(* IEC 61131-3 sources: repolevel_ST_code_completion/extract_code/重型运输系统/can/FUN, 13 files *)

(* ---- CAN_Read_Data_SWMC.st ---- *)
FUNCTION CAN_Read_Data_SWMC : Can_baseframe
VAR_INPUT
	SWMC_ID	 :UINT;		//接收SWMC控制ID
	I	 	 :UINT;      //接收缓冲区域
END_VAR
VAR
	frame :Can_baseframe;
END_VAR

CASE  SWMC_ID OF

	1:                       //SWMC-C1
		frame.id 	:= (gCan.C1RxMsg.RXMsg[I].RxMsg_CobId-8)/32;
		frame.data 	:= gCan.C1RxMsg.RXMsg[I].RxMsg_Byte;
	2:                       //SWMC-C2
		frame.id 	:= (gCan.C2RxMsg.RXMsg[I].RxMsg_CobId-8)/32;
		frame.data 	:= gCan.C2RxMsg.RXMsg[I].RxMsg_Byte;
	3:						//SWMC-C3
		frame.id 	:= (gCan.C3RxMsg.RXMsg[I].RxMsg_CobId-8)/32;
		frame.data 	:= gCan.C3RxMsg.RXMsg[I].RxMsg_Byte;
	4:                       //SWMC-C4
		frame.id 	:= (gCan.C4RxMsg.RXMsg[I].RxMsg_CobId-8)/32;
		frame.data 	:= gCan.C4RxMsg.RXMsg[I].RxMsg_Byte;
	//(*
	5:                       //SWMC-C5
		frame.id 	:= (gCan.C5RxMsg.RXMsg[I].RxMsg_CobId-8)/32;
		frame.data 	:= gCan.C5RxMsg.RXMsg[I].RxMsg_Byte;
	6:						//SWMC-C6
		frame.id 	:= (gCan.C6RxMsg.RXMsg[I].RxMsg_CobId-8)/32;
		frame.data 	:= gCan.C6RxMsg.RXMsg[I].RxMsg_Byte;
		//*)
	ELSE				//Other
		frame.id := 0;
		frame.data[1] := 0;
		frame.data[2] := 0;
		frame.data[3] := 0;
		frame.data[4] := 0;
		frame.data[5] := 0;
		frame.data[6] := 0;
		frame.data[7] := 0;
		frame.data[8] := 0;
END_CASE
Can_Read_data_SWMC := frame;

(* ---- CAN_Send_Data_SWMC.st ---- *)
FUNCTION CAN_Send_Data_SWMC : BOOL
VAR_INPUT
	SWMC_ID : UINT;
	id 		: UINT;
	data	: ARRAY[1..8] OF BYTE;
END_VAR
VAR

END_VAR

CASE  SWMC_ID OF

	1:
		gCan.C1TxMsg.TXMsg[1].TxMsg_CobId 	:= 8 + 32 * id;
	  	gCan.C1TxMsg.TXMsg[1].TxMsg_Byte 	:= data;
	   	gCan.C1TxMsg.NoOfTxMessages			:= 1;
	   	gCan.C1TxMsg.TxCounter 				:= gCan.C1TxMsg.TxCounter +1;
	2:
		gCan.C2TxMsg.TXMsg[1].TxMsg_CobId 	:= 8 + 32 * id;
	  	gCan.C2TxMsg.TXMsg[1].TxMsg_Byte 	:= data;
	   	gCan.C2TxMsg.NoOfTxMessages			:= 1;
	   	gCan.C2TxMsg.TxCounter 				:= gCan.C2TxMsg.TxCounter +1;
	3:
		gCan.C3TxMsg.TXMsg[1].TxMsg_CobId 	:= 8 + 32 * id;
	  	gCan.C3TxMsg.TXMsg[1].TxMsg_Byte 	:= data;
	   	gCan.C3TxMsg.NoOfTxMessages			:= 1;
	   	gCan.C3TxMsg.TxCounter 				:= gCan.C3TxMsg.TxCounter +1;
	4:
		gCan.C4TxMsg.TXMsg[1].TxMsg_CobId 	:= 8 + 32 * id;
	  	gCan.C4TxMsg.TXMsg[1].TxMsg_Byte 	:= data;
	   	gCan.C4TxMsg.NoOfTxMessages			:= 1;
	   	gCan.C4TxMsg.TxCounter 				:= gCan.C4TxMsg.TxCounter +1;
	//(*
	5:
		gCan.C5TxMsg.TXMsg[1].TxMsg_CobId 	:= 8 + 32 * id;
	  	gCan.C5TxMsg.TXMsg[1].TxMsg_Byte 	:= data;
	   	gCan.C5TxMsg.NoOfTxMessages			:= 1;
	   	gCan.C5TxMsg.TxCounter 				:= gCan.C5TxMsg.TxCounter +1;
	6:
		gCan.C6TxMsg.TXMsg[1].TxMsg_CobId 	:= 8 + 32 * id;
	  	gCan.C6TxMsg.TXMsg[1].TxMsg_Byte 	:= data;
	   	gCan.C6TxMsg.NoOfTxMessages			:= 1;
	   	gCan.C6TxMsg.TxCounter 				:= gCan.C6TxMsg.TxCounter +1;
	//*)

END_CASE

(* ---- percentCalc.st ---- *)
FUNCTION percentCalc : REAL
VAR_INPUT
	level		:INT;	//1->地轨	2->天轨
	idx			:INT;	//挡板索引编号
END_VAR
VAR
	c			:REAL;
	p			:REAL;
END_VAR

//伸出百分比计算
CASE level OF
	1:
		IF gDev.grd[idx].sensor.position < 3 THEN
			RETURN;
		END_IF
		c := gDev.grd[idx].sensor.position - gDev.grd[idx].sensor.retractVal;
		p := gDev.grd[idx].sensor.extendVal - gDev.grd[idx].sensor.retractVal;
		percentCalc := c * 100 / p;
	2:
		IF gDev.sky[idx].sensor.position < 3 THEN
			RETURN;
		END_IF
		c := gDev.sky[idx].sensor.position - gDev.sky[idx].sensor.retractVal;
		p := gDev.sky[idx].sensor.extendVal - gDev.sky[idx].sensor.retractVal;
		percentCalc := c * 100 / p;
END_CASE

(* ---- setButtonByDirect.st ---- *)
FUNCTION setButtonByDirect : BOOL
VAR_INPUT
	level		:INT;	//1->地轨	2->天轨
	idx			:INT;	//挡板索引编号
	direct		:TargetDirect;
END_VAR
VAR
END_VAR
//	本函数用于根据输入参数 操作UI界面的按钮变量
CASE level OF
	1:
		IF idx = 0 OR idx > 10 THEN		//参数校验
			RETURN;
		END_IF
		CASE direct OF
			TargetDirect.extend:
				gUI.grd[idx].btnStop := FALSE;
				gUI.grd[idx].btnExtend := TRUE;
				gUI.grd[idx].btnRetract := FALSE;
			TargetDirect.retract:
				gUI.grd[idx].btnStop := FALSE;
				gUI.grd[idx].btnExtend := FALSE;
				gUI.grd[idx].btnRetract := TRUE;
			TargetDirect.stop:
				gUI.grd[idx].btnStop := FALSE;
				gUI.grd[idx].btnExtend := FALSE;
				gUI.grd[idx].btnRetract := FALSE;
		END_CASE
	2:
		IF idx > 10 THEN		//参数校验
			RETURN;
		END_IF
		CASE direct OF
			TargetDirect.extend:
				gUI.sky[idx].btnStop := FALSE;
				gUI.sky[idx].btnExtend := TRUE;
				gUI.sky[idx].btnRetract := FALSE;
			TargetDirect.retract:
				gUI.sky[idx].btnStop := FALSE;
				gUI.sky[idx].btnExtend := FALSE;
				gUI.sky[idx].btnRetract := TRUE;
			TargetDirect.stop:
				gUI.sky[idx].btnStop := FALSE;
				gUI.sky[idx].btnExtend := FALSE;
				gUI.sky[idx].btnRetract := FALSE;
		END_CASE

END_CASE;

(* ---- updateDevStatus.st ---- *)
FUNCTION updateDevStatus : DevStatus
VAR_INPUT
	level		:INT;		//1->地轨	2->天轨
	idx			:INT;		//挡板索引编号
	errorVal	:REAL;		//误差范围
END_VAR
VAR
	extendVal	:REAL;		//伸出值
	retractVal	:REAL;		//缩回到位值
	nowVal		:REAL;		//当前值
	stat		:DevStatus;	//设备状态
END_VAR

(* 本函数用于根据设备的标定伸出/缩回值以及当前位置
** 判断该缸体是否处于伸出/缩回到位状态，如果到位更新参数
*)

stat := DevStatus.unknown;	//初始化状态量
CASE level OF
	1:
		extendVal := gDev.grd[idx].sensor.extendVal;
		retractVal := gDev.grd[idx].sensor.retractVal;
		nowVal := gDev.grd[idx].sensor.position;
		stat := gDev.grd[idx].state;
	2:
		extendVal := gDev.sky[idx].sensor.extendVal;
		retractVal := gDev.sky[idx].sensor.retractVal;
		nowVal := gDev.sky[idx].sensor.position;
		stat := gDev.sky[idx].state;
END_CASE

IF nowVal > 1 THEN
	IF nowVal < retractVal + errorVal THEN
		stat := DevStatus.retracted;
	ELSIF nowVal > extendVal - errorVal THEN
		stat := DevStatus.extended;
	ELSE
		IF stat <> DevStatus.runing THEN
			stat := DevStatus.error;
		END_IF
	END_IF
ELSE
	stat := DevStatus.unknown;
END_IF

CASE level OF
	1:
		gDev.grd[idx].state := stat;
	2:
		gDev.sky[idx].state := stat;
END_CASE

updateDevStatus := stat;

(* ---- CommandExecutor.st ---- *)
FUNCTION_BLOCK CommandExecutor
VAR_INPUT
	level		:INT;			//1->地轨	2->天轨
	idx			:INT;			//挡板索引编号
	percent		:REAL;			//比例阀百分比 传入-100~+100
END_VAR
VAR_OUTPUT
END_VAR
VAR
END_VAR

IF percent > 0 THEN
	CASE level OF
		1:
			gController.grd[idx].extendPercent := REAL_TO_WORD(percent * 65535 / 100);
			gController.grd[idx].retractPercent := 0;
		2:
			gController.sky[idx].extendPercent := REAL_TO_WORD(percent * 65535 / 100);
			gController.sky[idx].retractPercent := 0;
	END_CASE
ELSE
	CASE level OF
		1:
			gController.grd[idx].extendPercent := 0;
			gController.grd[idx].retractPercent := REAL_TO_WORD(ABS(percent) * 65535 / 100);
		2:
			gController.sky[idx].extendPercent := 0;
			gController.sky[idx].retractPercent := REAL_TO_WORD(ABS(percent) * 65535 / 100);
	END_CASE
END_IF

(* ---- CommandExecutor0.st ---- *)
FUNCTION_BLOCK CommandExecutor0
VAR_INPUT
	level		:INT;			//1->地轨	2->天轨
	idx			:INT;			//挡板索引编号
	direct		:TargetDirect;	//方向
	percent		:REAL;			//比例阀百分比 传入0-100
END_VAR
VAR_OUTPUT
END_VAR
VAR
END_VAR

CASE direct OF
	TargetDirect.extend:
		CASE level OF
			1:
				gController.grd[idx].extendPercent := REAL_TO_WORD(percent * 65535 / 100);
				gController.grd[idx].retractPercent := 0;
			2:
				gController.sky[idx].extendPercent := REAL_TO_WORD(percent * 65535 / 100);
				gController.sky[idx].retractPercent := 0;
		END_CASE
	TargetDirect.retract:
		CASE level OF
			1:
				gController.grd[idx].extendPercent := 0;
				gController.grd[idx].retractPercent := REAL_TO_WORD(percent * 65535 / 100);
			2:
				gController.sky[idx].extendPercent := 0;
				gController.sky[idx].retractPercent := REAL_TO_WORD(percent * 65535 / 100);
		END_CASE
	TargetDirect.stop:
		CASE level OF
			1:
				gController.grd[idx].extendPercent := 0;
				gController.grd[idx].retractPercent := 0;
			2:
				gController.sky[idx].extendPercent := 0;
				gController.sky[idx].retractPercent := 0;
		END_CASE

	ELSE
		CASE level OF
			1:
				gController.grd[idx].extendPercent := 0;
				gController.grd[idx].retractPercent := 0;
			2:
				gController.sky[idx].extendPercent := 0;
				gController.sky[idx].retractPercent := 0;
		END_CASE

END_CASE

(* ---- fileSave.st ---- *)
FUNCTION_BLOCK fileSave
VAR_INPUT
	filePath 	:STRING;
	intervalt	:INT;
END_VAR
VAR
	lineCount	: INT;
	fileHandle  : DWORD;
	fileName	: STRING;
END_VAR
VAR_OUTPUT
END_VAR

(* ---- fileSave_close.st ---- *)
FUNCTION_BLOCK fileSave
VAR_INPUT
	filePath 	:STRING;
	intervalt	:INT;
END_VAR
VAR
	lineCount	: INT;
	fileHandle  : DWORD;
	fileName	: STRING;
END_VAR
VAR_OUTPUT
END_VAR

IF fileHandle <> 0 THEN
	SysFileClose(hFile := fileHandle);
	fileHandle := 0;
END_IF

(* ---- fileSave_createDir.st ---- *)
FUNCTION_BLOCK fileSave
VAR_INPUT
	filePath 	:STRING;
	devName		: STRING ;
	intervalt	:INT;
END_VAR
VAR
	lineCount	: INT;
	fileHandle  : DWORD;
	fileName	: STRING;
	filePath1	:STRING;
END_VAR
VAR_OUTPUT
END_VAR

filePath1 := FilePath;
filePath1 := concat(filePath1,'/');
filePath1 := concat(filePath1,devName);
SysDirCreate2(filePath1, TRUE);

(* ---- fileSave_new.st ---- *)
FUNCTION_BLOCK fileSave
VAR_INPUT
	filePath 	:STRING;
	intervalt	:INT;
	devName		: STRING ;
END_VAR
VAR
	lineCount	: INT;
	fileHandle  : DWORD;
	fileName	: STRING;
	fileHandle0 : DWORD;
	datetime	: DATE_AND_TIME;
	UdIntms 	: UDINT;
	UdMsOffset  : UDINT;
	DTimer_Str  : STRING;
	uiYear 		: UINT;
    uiMonth 	: UINT;
    uiDay 		: UINT;
    uiHour 		: UINT;
    uiMinute 	: UINT;
    uiSecond 	: UINT;
	uiMsSecond	: UINT;

	S_Time64		:  SysTime64;
	STT			:  CurTimeEx;
	S_Time			:  SystemTimeDate;
	Time_Str		:  STRING;
	F_err		: DWORD;
	F_HANDL		: DWORD;
END_VAR
VAR_OUTPUT
END_VAR

	STT(SystemTime:= S_Time64, TimeDate:= S_Time);
	Time_Str :='';
	Time_Str := concat(Time_Str,UINT_TO_STRING(S_Time.Year));
	Time_Str := concat(Time_Str,'-');
	Time_Str := concat(Time_Str,UINT_TO_STRING(S_Time.Month));
	Time_Str := concat(Time_Str,'-');
	Time_Str := concat(Time_Str,UINT_TO_STRING(S_Time.Day));
	Time_Str := concat(Time_Str,'_');
	Time_Str := concat(Time_Str,UINT_TO_STRING(S_Time.Hour));
	Time_Str := concat(Time_Str,'-');
	Time_Str := concat(Time_Str,UINT_TO_STRING(S_Time.Minute));
	Time_Str := concat(Time_Str,'-');
	Time_Str := concat(Time_Str,UINT_TO_STRING(S_Time.Second));
	Time_Str := concat(Time_Str,'_');
	Time_Str := concat(Time_Str,UINT_TO_STRING(S_Time.Milliseconds));

	fileName := FilePath;
	fileName := concat(fileName,'/');
	fileName := concat(fileName,devName);

	fileName := concat(fileName,'/');
	fileName := concat(fileName,devName);
	fileName := concat(fileName,'-');
	fileName := concat(fileName,Time_Str);
    fileName := concat(fileName,'.txt');

	fileHandle := SysFileOpen(szFile:= fileName, am:=ACCESS_MODE.AM_WRITE, pResult:= ADR(F_err));
	lineCount := -1;
	//fileHandle := SysFileOpen(szFile:= fileName, am:=ACCESS_MODE.AM_APPEND, pResult:= ADR(F_err));

(* ---- fileSave_write.st ---- *)
FUNCTION_BLOCK fileSave
VAR_INPUT
	filePath 	:STRING;
	intervalt	:INT;
	positionInt 	:INT;
	speedInt 		:INT;
	stateInt		:INT;
END_VAR
VAR
	lineCount	: INT;
	fileHandle  : DWORD;
	fileName	: STRING;
	data		: STRING;
	F_err		: DWORD;
	tempInt		: INT;
END_VAR
VAR_OUTPUT
END_VAR

IF fileHandle <> 0 THEN
	lineCount := lineCount + 1;
	tempInt	:= lineCount * intervalt;
	data := INT_TO_STRING(lineCount);
	data := concat(data,'$T$T');
	data := concat(data, INT_TO_STRING(tempInt));
	IF tempInt < 1000 THEN
		data := concat(data,'$T');
	END_IF
	data := concat(data,'$T$T');
	data := concat(data,INT_TO_STRING(positionInt));
	data := concat(data,'$T');
	data := concat(data,INT_TO_STRING(speedInt));
	data := concat(data,'$T');
	data := concat(data,INT_TO_STRING(stateInt));
	data := concat(data,'$R');

	SysFileWrite(hFile:=fileHandle , pbyBuffer:= ADR(data) , ulSize:= DINT_TO_DWORD(SysStrLen(data)) , pResult:= ADR(F_err));		// 写入数据

END_IF

(* ---- tcpUpload_send.st ---- *)
FUNCTION_BLOCK tcpUpload
VAR_INPUT
	InetAddress		:STRING;
	port			:UINT;
	dataLength		:__XINT;
	sendBuf 		:ARRAY[1..1024]OF BYTE;
END_VAR
VAR_OUTPUT
END_VAR
VAR
	tcpConnector	:TCP.Connector;
	tcpStream		:TCP.Stream;
	pointerStream	:POINTER TO TCP.Stream;
	sizeData		:__XINT;

	tcpState		:UINT:=0;
	tcpCount		:UINT:=0;

	netState		:INT;
END_VAR

tcpCount := tcpCount + 1;
CASE tcpState OF

	0:			//connet server
		tcpConnector.Connect(sIPAddress:= InetAddress,uiPort:= port,pStream => pointerStream);
		IF pointerStream<>0 THEN
			tcpState :=1;
		ELSE
			tcpState :=2;
		END_IF

	1:
		netState := pointerStream^.Send(ADR(sendBuf),dataLength,diSent=>sizeData);
		IF netState <> 0 THEN
			tcpState := 2;
		END_IF

	2:		 	//断开连接
	    tcpConnector.Disconnect();
		tcpState := 0;

END_CASE
